PROGRAM Transfer
VAR
	nSource: INT;
	nDestination: INT;
	bTransferStartTime : BOOL;
	nStartTimeInSeconds :UDINT;
	nTime: UDINT;
	
	tempSecondsToAddWhilePause: DINT;
	SecondsToAddWhilePause: DINT;
	
	RemainingTime: UDINT;
	fbRTRIG: R_TRIG;
	fbRTRIGEnable : BOOL;
	fbRTRIG2: F_TRIG;
	fbRTRIG2Enable : BOOL;


	fbFTRIGLLS : F_TRIG;
	fbFTRIGLLSEnable : BOOL;
	fbFTRIGLLS2 : F_TRIG;
	fbFTRIGLLS2Enable : BOOL;
	fbFTRIGULS : F_TRIG;
	fbFTRIGULSEnable : BOOL;
	bCommandToPumpStart:BOOL;
	fbSelection : FBSelection;

	
	bStartCommand: BOOL;
	CLK: INT;
	Q: INT;
	btransferBlockEnded: BOOL;
	
	sSourceName: STRING;
	sDestinationName: STRING;
	bMode: BOOL;
	
	DestinationULSON: BOOL;
END_VAR

VAR_INPUT	
	nCurrentBlock : INT;
END_VAR

// RECEIVE SOURCE , DESTINATION AND MODE INFORMATION FROM THE BLOCK //

sSourceName:= RecipeTags.Recipe.Blocks[nCurrentBlock].Properties.sSource;
sDestinationName:=RecipeTags.Recipe.Blocks[nCurrentBlock].Properties.sDestination;
bMode := RecipeTags.Recipe.Blocks[nCurrentBlock].Properties.bModeSelection;

// Converting Names to NUmbers FROM HELPERS/VESSEL SELECTION.FBSELECTION.TARGETCONVERTER //

fbSelection.TargetConverter(sTargetName:= sSourceName, TargetConverter_output => nSource); 
fbSelection.TargetConverter(sTargetName:=sDestinationName, TargetConverter_output=>nDestination);






IF nSource<9 THEN
	fbFTRIGLLS(CLK:=IO.Vessels[nSource].LLS);
END_IF


IF nDestination<9 THEN
	DestinationULSON := Not(IO.Vessels[nDestination].ULS);

//ELSIF nDestination>=9 AND nDestination<=11 THEN
//	fbFTRIGLLS2(CLK:=IO.Vessels[nSource].LLS);
//	IF fbFTRIGLLS2.Q THEN
//		DestinationULSON := TRUE;
//	ELSE
//		DestinationULSON := FALSE;
//	END_IF
ELSE
	DestinationULSON :=  FALSE;
END_IF



IF fbFTRIGLLS.Q THEN
	fbFTRIGLLSEnable := TRUE;
END_IF


IF nSource=12 THEN
	fbRTRIG2(CLK:=IO.Vessels[nDestination].ULS);
END_IF



IF fbRTRIG2.Q THEN
	fbRTRIG2Enable := TRUE;
	RecipeTags.bBlockStart[nCurrentBlock] := FALSE;
END_IF	





// Start Time - Writing start time to structure //

IF (bTransferStartTime=FALSE) THEN
	RecipeTags.Recipe.Blocks[nCurrentBlock].Properties.sStartTime:=MAIN.sConcatenatedHourMinuteString;
	nStartTimeInSeconds:= STRING_TO_UDINT(MAIN.sCurrentSecond);
	bTransferStartTime:=  TRUE;
END_IF

// Time Intervals - Conversion of input time as per selection//

IF RecipeTags.Recipe.Blocks[nCurrentBlock].Properties.sIntervalType = 'S' THEN
	nTime := DINT_TO_UDINT(RecipeTags.Recipe.Blocks[nCurrentBlock].Properties.nInterval);
ELSIF RecipeTags.Recipe.Blocks[nCurrentBlock].Properties.sIntervalType = 'M' THEN
	nTime := DINT_TO_UDINT(RecipeTags.Recipe.Blocks[nCurrentBlock].Properties.nInterval * 60);
ELSIF RecipeTags.Recipe.Blocks[nCurrentBlock].Properties.sIntervalType = 'H' THEN
	nTime := DINT_TO_UDINT(RecipeTags.Recipe.Blocks[nCurrentBlock].Properties.nInterval * 3600);
END_IF

// Track time elapsed for resume when pause is released //

IF RecipeTags.enWaitPause[nCurrentBlock] THEN
	tempSecondsToAddWhilePause := tempSecondsToAddWhilePause + 1;
	SecondsToAddWhilePause := tempSecondsToAddWhilePause; 
ELSE
	tempSecondsToAddWhilePause := 0;
	SecondsToAddWhilePause :=0;
END_IF

// TO CHECK BLOCK START //

IF NOT(RecipeTags.bPauseRecipe) THEN
		RecipeTags.enWaitPause[nCurrentBlock] := FALSE;
		RecipeTags.bBlockStart[nCurrentBlock] := TRUE;
		//IF bmode THEN
		//	RemainingTime := ABS(nTime- nStartTimeInSeconds-STRING_TO_UDINT(MAIN.sCurrentSecond));
		//ELSE
		//	RemainingTime := 0;
		//END_IF
ELSE
		RecipeTags.bBlockStart[nCurrentBlock] := FALSE;
		RecipeTags.enWaitPause[nCurrentBlock] := TRUE;
END_IF

// TO CHECK BLOCK COMPLETION  //

IF bmode THEN
	// time based mode //
	IF  (nTime + nStartTimeInSeconds + DINT_TO_UDINT(TRUNC(SecondsToAddWhilePause/100))) 
		          <= (STRING_TO_UDINT(MAIN.sCurrentSecond)) OR DestinationULSON  OR fbRTRIG2Enable THEN
		RecipeTags.Recipe.Blocks[nCurrentBlock].Properties.bStopCommand := TRUE;
		RecipeTags.Recipe.Blocks[nCurrentBlock].Properties.sEndTime:=MAIN.sConcatenatedHourMinuteString;
		RecipeTags.bBlockStart[nCurrentBlock] := FALSE;
		RecipeTags.bBlockEnd[nCurrentBlock] := TRUE;
		fbFTRIGLLSEnable := FALSE;
		fbRTRIG2Enable := FALSE;
		
	ELSE
		RecipeTags.bBlockEnd[nCurrentBlock] := FALSE;
	END_IF
ELSE
	// level based mode //
	RecipeTags.bBlockEnd[nCurrentBlock] := FALSE;
	IF DestinationULSON OR fbRTRIG2Enable OR (fbFTRIGLLSEnable AND nDestination>=9 AND nDestination<12 ) THEN
		EndLogic(nCurrentBlock:=RecipeTags.bBlockEnd[nCurrentBlock]); 
		RecipeTags.bBlockEnd[nCurrentBlock] := TRUE;
		RecipeTags.bBlockStart[nCurrentBlock] := FALSE;
		fbFTRIGLLSEnable := FALSE;
		fbRTRIG2Enable := FALSE;
	END_IF
END_IF



ActivationLogic(nCurrentBlock:= nCurrentBlock, nSource:=nSource, nDestination:=nDestination);

   // IF BLOCK END HAS BEEN MADE TRUE //
EndLogic(nCurrentBlock:=RecipeTags.bBlockEnd[nCurrentBlock]);
IF EndLogic.OutputBool THEN
	fbRTRIGEnable := TRUE;
	RecipeTags.bBlockStart[nCurrentBlock] :=FALSE;
	EndLogic(nCurrentBlock:=RecipeTags.bBlockEnd[nCurrentBlock]);
END_IF

IF ((fbRTRIGEnable AND NOT(RecipeTags.bRuntimeEdit))  AND RecipeTags.Recipe.Blocks[nCurrentBlock].Name = 'Transfer') THEN
	ActivationLogic(nCurrentBlock:= nCurrentBlock, nSource:=nSource, nDestination:=nDestination);
	SecondsToAddWhilePause := 0;
	fbRTRIGEnable := FALSE;
	nTime := 0;
	bTransferStartTime := FALSE;
	//nStartTimeInSeconds := 0;
	RecipeTags.bBlockStart[nCurrentBlock]  :=FALSE;
	RecipeTags.bStartTimeEnable[nCurrentBlock] := FALSE;
	RecipeTags.bBlockEnd[nCurrentBlock] := FALSE;
//	EndLogic(nCurrentBlock:=RecipeTags.bBlockEnd[nCurrentBlock]);
	RecipeTags.bStartTimeEnable[nCurrentBlock] :=  FALSE;
	RecipeTags.Recipe.Blocks[nCurrentBlock].Properties.sEndTime:=MAIN.sConcatenatedHourMinuteString;
	RecipeTags.Recipe.Blocks[nCurrentBlock].Properties.bStopCommand := TRUE;
	

END_IF

END_PROGRAM

(* stored: Version 1.1.0.1, ProductVersion 3.1.4024.5
   POU Transfer: Id {3c5090f8-8148-4616-b5f6-620b86144fac}, SpecialFunc None *)
